TYPE "OOAx_Alr"
VERSION : 0.1
// Block: OOAx_Alr
   STRUCT
      TargetPosIncorrect : Bool;
      PosOutTolerance : Bool;
      WrongDirection : Bool;
      WrongNotIncrease : Bool;
      HwLimitMinus : Bool;
      HwLimitPlus : Bool;
      TimeoutPreset : Bool;
   END_STRUCT;

END_TYPE
